KUKA KRL program: prueba_gewindebolzen_.src, prueba_gewindebolzen_.dat

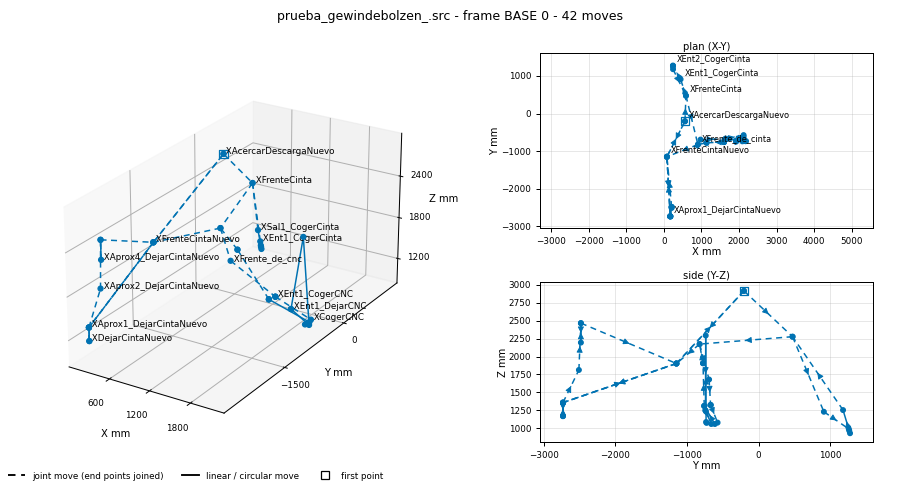
[picture p0: tool path of prueba_gewindebolzen_.src in frame BASE 0, 42 of 44 moves have a stored position in this frame; points joined in program order, loops and branches not executed]
--- prueba_gewindebolzen_.src ---
&ACCESS RVP
&REL 19
&COMMENT M36x315+allen
&PARAM TEMPLATE = C:\KRC\Roboter\Template\vorgabe
&PARAM EDITMASK = *
DEF prueba_gewindebolzen_( )
;FOLD INI;%{PE}%V3.2.0,%MKUKATPBASIS,%CINIT,%VCOMMON,%P
;FOLD BAS INI;%{E}%V3.2.0,%MKUKATPBASIS,%CINIT,%VINIT,%P
GLOBAL INTERRUPT DECL 3 WHEN $STOPMESS==TRUE DO IR_STOPM ( )
INTERRUPT ON 3
BAS (#INITMOV,0 )
;ENDFOLD (BAS INI)
;FOLD A20 INI;%{E}%V3.2.0,%MKUKATPA20,%CINIT,%VINIT,%P
IF ARC20==TRUE THEN
A20 (ARC_INI)
INTERRUPT DECL 6 WHEN $CYCFLAG[3]==FALSE DO A20(TECH_STOP2)
ENDIF
;ENDFOLD (A20 INI)
;FOLD A10 INI;%{E}%V3.2.0,%MKUKATPARC,%CINIT,%VINIT,%P
IF A10_OPTION==#ACTIVE THEN
INTERRUPT DECL 4 WHEN $CYCFLAG[2]==FALSE DO A10 (#APPL_ERROR)
INTERRUPT DECL 7 WHEN A_ARC_SWI==#ACTIVE DO A10 (#ARC_SEAM)
INTERRUPT DECL 5 WHEN A_FLY_ARC==TRUE DO A10 (#HPU_ARC)
INTERRUPT  ON 5
A10_INI ( )
ENDIF
;ENDFOLD (A10 INI)
;FOLD GRIPPER INI;%{E}%V3.2.0,%MKUKATPGRIPPER,%CINIT,%VINIT,%P
USER_GRP(0,DUMMY,DUMMY,GDEFAULT)
;ENDFOLD (GRIPPER INI)
;FOLD SPOT INI;%{E}%V3.2.0,%MKUKATPSPOT,%CINIT,%VINIT,%P
USERSPOT(#INIT)
;ENDFOLD (SPOT INI)
;FOLD TOUCHSENSE INI;%{E}%V3.2.0,%MKUKATPTS,%CINIT,%VINIT,%P
IF H70_OPTION THEN
INTERRUPT DECL 15 WHEN $MEAS_PULSE[TOUCH_I[TOUCH_ACTIVE].IN_NR] DO H70 (6,CD0 )
INTERRUPT DECL 16 WHEN $ZERO_MOVE DO H70 (7,CD0 )
INTERRUPT DECL 17 WHEN $TECHPAR_C[FG_TOUCH,8]>0.5 DO H70 (8,CD0)
H70 (1,CD0 )
ENDIF
;ENDFOLD (TOUCHSENSE INI)
;FOLD USER INI;%{E}%V3.2.0,%MKUKATPUSER,%CINIT,%VINIT,%P
;Make your modifications here
;ENDFOLD (USER INI)
;ENDFOLD (INI)

;=========================================================
;                Gewindebolzen
;       M36x315 Allen 16 + previo longitud 93
;                Codigo 257152360315
;
;=========================================================

;FOLD INICIALIZACION

INTERRUPT DECL 20 WHEN $IN[20]==FALSE DO PARO()
INTERRUPT OFF 20
;FOLD WAIT FOR IN 20 'InAire'  State= TRUE ;%{PE}%R 4.1.7,%MKUKATPBASIS,%CWAIT_FOR,%VWAIT_FOR,%P 1:0, 2:20, 3:'InAire', 5:TRUE, 6:
WAIT FOR $IN[20]==TRUE
;ENDFOLD


;FOLD PTP HOME CONT Vel= 5 % PDAT1;%{PE}%R 4.1.7,%MKUKATPBASIS,%CMOVE,%VPTP,%P 1:PTP, 2:HOME, 3:C_PTP, 5:5, 7:PDAT1
$BWDSTART = FALSE
PDAT_ACT=PPDAT1
BAS(#PTP_DAT)
FDAT_ACT=FHOME
BAS(#FRAMES)
BAS(#VEL_PTP,5)
$H_POS=XHOME
PTP XHOME C_PTP
;ENDFOLD
;FOLD WAIT Time=0 sec;%{PE}%R 5.5.32,%MKUKATPBASIS,%CWAIT,%VWAIT,%P 2:0
WAIT SEC 0
;ENDFOLD
DELMENS()


INTERRUPT ON 20

;$OV_PRO=nVeloFuera

bMarchaCintaSuperior=FALSE
bRobotEnCintaSup=FALSE
;FOLD OUT 1 'OutMarchaCintaSup'  State= FALSE CONT;%{PE}%R 4.1.7,%MKUKATPBASIS,%COUT,%VOUTX,%P 2:1, 3:'OutMarchaCintaSup', 5:FALSE, 6:CONTINUE
CONTINUE
$OUT[1]=FALSE
;ENDFOLD
;FOLD OUT 2 'OutMarchaCNC'  State= FALSE CONT;%{PE}%R 4.1.7,%MKUKATPBASIS,%COUT,%VOUTX,%P 2:2, 3:'OutMarchaCNC', 5:FALSE, 6:CONTINUE
CONTINUE
$OUT[2]=FALSE
;ENDFOLD
;FOLD OUT 3 'OutRobotDentroCNC'  State= FALSE CONT;%{PE}%R 4.1.7,%MKUKATPBASIS,%COUT,%VOUTX,%P 2:3, 3:'OutRobotDentroCNC', 5:FALSE, 6:CONTINUE
CONTINUE
$OUT[3]=FALSE
;ENDFOLD
;FOLD OUT 7 'OutRobotFuerCNC'  State= TRUE CONT;%{PE}%R 4.1.7,%MKUKATPBASIS,%COUT,%VOUTX,%P 2:7, 3:'OutRobotFuerCNC', 5:TRUE, 6:CONTINUE
CONTINUE
$OUT[7]=TRUE
;ENDFOLD
;FOLD OUT 8 'OutAbrirPlatoCNC'  State= FALSE CONT;%{PE}%R 4.1.7,%MKUKATPBASIS,%COUT,%VOUTX,%P 2:8, 3:'OutAbrirPlatoCNC', 5:FALSE, 6:CONTINUE
CONTINUE
$OUT[8]=FALSE
;ENDFOLD
;FOLD OUT 9 'OutCerrarPlatoCNC'  State= FALSE CONT;%{PE}%R 4.1.7,%MKUKATPBASIS,%COUT,%VOUTX,%P 2:9, 3:'OutCerrarPlatoCNC', 5:FALSE, 6:CONTINUE
CONTINUE
$OUT[9]=FALSE
;ENDFOLD
;FOLD OUT 10 'OutAvanContrpuntoCNC'  State= FALSE CONT;%{PE}%R 4.1.7,%MKUKATPBASIS,%COUT,%VOUTX,%P 2:10, 3:'OutAvanContrpuntoCNC', 5:FALSE, 6:CONTINUE
CONTINUE
$OUT[10]=FALSE
;ENDFOLD
;FOLD OUT 11 'OutRetroContrpuntoCNC'  State= FALSE CONT;%{PE}%R 4.1.7,%MKUKATPBASIS,%COUT,%VOUTX,%P 2:11, 3:'OutRetroContrpuntoCNC', 5:FALSE, 6:CONTINUE
CONTINUE
$OUT[11]=FALSE
;ENDFOLD
;FOLD OUT 12 'OutAbrirLunetaCNC'  State= FALSE CONT;%{PE}%R 4.1.7,%MKUKATPBASIS,%COUT,%VOUTX,%P 2:12, 3:'OutAbrirLunetaCNC', 5:FALSE, 6:CONTINUE
CONTINUE
$OUT[12]=FALSE
;ENDFOLD
;FOLD OUT 17 'OutCerrarLunetaCNC'  State= FALSE CONT;%{PE}%R 4.1.7,%MKUKATPBASIS,%COUT,%VOUTX,%P 2:17, 3:'OutCerrarLunetaCNC', 5:FALSE, 6:CONTINUE
CONTINUE
$OUT[17]=FALSE
;ENDFOLD


bParadaManiobra=FALSE
;FOLD WAIT FOR ( IN 4 'InPulsadorMarcha' );%{PE}%R 5.5.33,%MKUKATPBASIS,%CEXT_WAIT_FOR,%VEXT_WAIT_FOR,%P 2:, 4:, 5:$IN, 6:4, 7:InPulsadorMarcha, 9:
WAIT FOR  ( $IN[4] )
;ENDFOLD
bMarchaCintaSuperior=TRUE
;FOLD WAIT Time=0.5 sec;%{PE}%R 5.5.33,%MKUKATPBASIS,%CWAIT,%VWAIT,%P 2:0.5
WAIT SEC 0.5
;ENDFOLD
bMarchaCintaSuperior=FALSE
;FOLD WAIT FOR NOT ( IN 4 'InPulsadorMarcha' );%{PE}%R 5.5.33,%MKUKATPBASIS,%CEXT_WAIT_FOR,%VEXT_WAIT_FOR,%P 2:NOT, 4:, 5:$IN, 6:4, 7:InPulsadorMarcha, 9:
WAIT FOR  NOT ( $IN[4] )
;ENDFOLD
outPilotoMarcha=TRUE

;------Soltar Piezas sobre Cinta de Descarga-------
IF ((InPinza1Abierta==FALSE) OR (InPinza2Abierta==FALSE)) THEN


;FOLD PTP AcercarDescargaNuevo CONT Vel= 30 % PDAT28 Tool[0] Base[0];%{PE}%R 4.1.16,%MKUKATPBASIS,%CMOVE,%VPTP,%P 1:PTP, 2:AcercarDescargaNuevo, 3:C_PTP, 5:30, 7:PDAT28
$BWDSTART = FALSE
PDAT_ACT=PPDAT28
BAS(#PTP_DAT)
FDAT_ACT=FAcercarDescargaNuevo
BAS(#FRAMES)
BAS(#VEL_PTP,30)
PTP XAcercarDescargaNuevo C_PTP
;ENDFOLD

;FOLD PTP FrenteCintaNuevo CONT Vel= 30 % PDAT26 Tool[0] Base[0];%{PE}%R 4.1.16,%MKUKATPBASIS,%CMOVE,%VPTP,%P 1:PTP, 2:FrenteCintaNuevo, 3:C_PTP, 5:30, 7:PDAT26
$BWDSTART = FALSE
PDAT_ACT=PPDAT26
BAS(#PTP_DAT)
FDAT_ACT=FFrenteCintaNuevo
BAS(#FRAMES)
BAS(#VEL_PTP,30)
PTP XFrenteCintaNuevo C_PTP
;ENDFOLD

;FOLD PTP Aprox1_DejarCintaNuevo CONT Vel= 30 % PDAT27 Tool[2]:Tool2      Base[0];%{PE}%R 4.1.16,%MKUKATPBASIS,%CMOVE,%VPTP,%P 1:PTP, 2:Aprox1_DejarCintaNuevo, 3:C_PTP, 5:30, 7:PDAT27
$BWDSTART = FALSE
PDAT_ACT=PPDAT27
BAS(#PTP_DAT)
FDAT_ACT=FAprox1_DejarCintaNuevo
BAS(#FRAMES)
BAS(#VEL_PTP,30)
PTP XAprox1_DejarCintaNuevo C_PTP
;ENDFOLD

;FOLD LIN DejarCintaNuevo CONT Vel= 0.3 m/s CPDAT1 Tool[2]:Tool2      Base[0];%{PE}%R 4.1.16,%MKUKATPBASIS,%CMOVE,%VLIN,%P 1:LIN, 2:DejarCintaNuevo, 3:C_DIS, 5:0.3, 7:CPDAT1
$BWDSTART = FALSE
LDAT_ACT=LCPDAT1
BAS(#CP_DAT)
FDAT_ACT=FDejarCintaNuevo
BAS(#FRAMES)
BAS(#VEL_CP,0.3)
LIN XDejarCintaNuevo C_DIS
;ENDFOLD

;FOLD SET Pinza2  State= OPN  Abrir;%{PE}%R 4.1.4,%MKUKATPGRP,%CGRP,%VGRP,%P 2:2, 4:1, 5:#NO, 6:Abrir, 8:0, 10:1
H50(GRP,2,1,GAbrir)
;ENDFOLD

;FOLD PTP Aprox1_DejarCintaNuevo CONT Vel= 30 % PDAT27 Tool[2]:Tool2      Base[0];%{PE}%R 4.1.16,%MKUKATPBASIS,%CMOVE,%VPTP,%P 1:PTP, 2:Aprox1_DejarCintaNuevo, 3:C_PTP, 5:30, 7:PDAT27
$BWDSTART = FALSE
PDAT_ACT=PPDAT27
BAS(#PTP_DAT)
FDAT_ACT=FAprox1_DejarCintaNuevo
BAS(#FRAMES)
BAS(#VEL_PTP,30)
PTP XAprox1_DejarCintaNuevo C_PTP
;ENDFOLD

;FOLD PTP Aprox2_DejarCintaNuevo CONT Vel= 30 % PDAT29 Tool[2]:Tool2      Base[0];%{PE}%R 4.1.16,%MKUKATPBASIS,%CMOVE,%VPTP,%P 1:PTP, 2:Aprox2_DejarCintaNuevo, 3:C_PTP, 5:30, 7:PDAT29
$BWDSTART = FALSE
PDAT_ACT=PPDAT29
BAS(#PTP_DAT)
FDAT_ACT=FAprox2_DejarCintaNuevo
BAS(#FRAMES)
BAS(#VEL_PTP,30)
PTP XAprox2_DejarCintaNuevo C_PTP
;ENDFOLD

;FOLD PTP Aprox3_DejarCintaNuevo CONT Vel= 30 % PDAT30 Tool[2]:Tool2      Base[0];%{PE}%R 4.1.16,%MKUKATPBASIS,%CMOVE,%VPTP,%P 1:PTP, 2:Aprox3_DejarCintaNuevo, 3:C_PTP, 5:30, 7:PDAT30
$BWDSTART = FALSE
PDAT_ACT=PPDAT30
BAS(#PTP_DAT)
FDAT_ACT=FAprox3_DejarCintaNuevo
BAS(#FRAMES)
BAS(#VEL_PTP,30)
PTP XAprox3_DejarCintaNuevo C_PTP
;ENDFOLD

;FOLD LIN Aprox4_DejarCintaNuevo CONT Vel= 0.3 m/s CPDAT13 Tool[2]:Tool2      Base[0];%{PE}%R 4.1.16,%MKUKATPBASIS,%CMOVE,%VLIN,%P 1:LIN, 2:Aprox4_DejarCintaNuevo, 3:C_DIS, 5:0.3, 7:CPDAT13
$BWDSTART = FALSE
LDAT_ACT=LCPDAT13
BAS(#CP_DAT)
FDAT_ACT=FAprox4_DejarCintaNuevo
BAS(#FRAMES)
BAS(#VEL_CP,0.3)
LIN XAprox4_DejarCintaNuevo C_DIS
;ENDFOLD

;FOLD SET Pinza1  State= OPN  Abrir;%{PE}%R 4.1.4,%MKUKATPGRP,%CGRP,%VGRP,%P 2:1, 4:1, 5:#NO, 6:Abrir, 8:0, 10:1
H50(GRP,1,1,GAbrir)
;ENDFOLD

;FOLD PTP Aprox3_DejarCintaNuevo CONT Vel= 30 % PDAT30 Tool[2]:Tool2      Base[0];%{PE}%R 4.1.16,%MKUKATPBASIS,%CMOVE,%VPTP,%P 1:PTP, 2:Aprox3_DejarCintaNuevo, 3:C_PTP, 5:30, 7:PDAT30
$BWDSTART = FALSE
PDAT_ACT=PPDAT30
BAS(#PTP_DAT)
FDAT_ACT=FAprox3_DejarCintaNuevo
BAS(#FRAMES)
BAS(#VEL_PTP,30)
PTP XAprox3_DejarCintaNuevo C_PTP
;ENDFOLD

;FOLD PTP FrenteCintaNuevo CONT Vel= 30 % PDAT26 Tool[0] Base[0];%{PE}%R 4.1.16,%MKUKATPBASIS,%CMOVE,%VPTP,%P 1:PTP, 2:FrenteCintaNuevo, 3:C_PTP, 5:30, 7:PDAT26
$BWDSTART = FALSE
PDAT_ACT=PPDAT26
BAS(#PTP_DAT)
FDAT_ACT=FFrenteCintaNuevo
BAS(#FRAMES)
BAS(#VEL_PTP,30)
PTP XFrenteCintaNuevo C_PTP
;ENDFOLD

;FOLD PTP AcercarDescargaNuevo CONT Vel= 30 % PDAT28 Tool[0] Base[0];%{PE}%R 4.1.16,%MKUKATPBASIS,%CMOVE,%VPTP,%P 1:PTP, 2:AcercarDescargaNuevo, 3:C_PTP, 5:30, 7:PDAT28
$BWDSTART = FALSE
PDAT_ACT=PPDAT28
BAS(#PTP_DAT)
FDAT_ACT=FAcercarDescargaNuevo
BAS(#FRAMES)
BAS(#VEL_PTP,30)
PTP XAcercarDescargaNuevo C_PTP
;ENDFOLD

ELSE

ENDIF

LOOP


;FOLD CHECK Pinza1  State= OPN  at START  Delay= 0 ms;%{PE}%R 4.1.4,%MKUKATPGRP,%CCHK_GRP,%VCHK_GRP,%P 2:1, 4:1, 6:0, 8:0
TRIGGER WHEN DISTANCE=0 DELAY=0 DO H50(CHK_APO_UP,1,1,GCONT)  PRIO=-1
;ENDFOLD
;FOLD CHECK Pinza2  State= OPN  at START  Delay= 0 ms;%{PE}%R 4.1.4,%MKUKATPGRP,%CCHK_GRP,%VCHK_GRP,%P 2:2, 4:1, 6:0, 8:0
TRIGGER WHEN DISTANCE=0 DELAY=0 DO H50(CHK_APO_UP,2,1,GCONT)  PRIO=-1
;ENDFOLD

;FOLD WAIT FOR IN 21 'InPinza1Abierta'  State= TRUE ;%{PE}%R 4.1.7,%MKUKATPBASIS,%CWAIT_FOR,%VWAIT_FOR,%P 1:0, 2:21, 3:'InPinza1Abierta', 5:TRUE, 6:
WAIT FOR $IN[21]==TRUE
;ENDFOLD
;FOLD WAIT FOR IN 23 'InPinza2Abierta'  State= TRUE ;%{PE}%R 4.1.7,%MKUKATPBASIS,%CWAIT_FOR,%VWAIT_FOR,%P 1:0, 2:23, 3:'InPinza2Abierta', 5:TRUE, 6:
WAIT FOR $IN[23]==TRUE
;ENDFOLD
;ENDFOLD


;FOLD COGER PIEZA DE CINTA

;FOLD PTP FrenteCinta CONT Vel= 30 % PDAT1 Tool[0] Base[0];%{PE}%R 4.1.7,%MKUKATPBASIS,%CMOVE,%VPTP,%P 1:PTP, 2:FrenteCinta, 3:C_PTP, 5:30, 7:PDAT1
$BWDSTART = FALSE
PDAT_ACT=PPDAT1
BAS(#PTP_DAT)
FDAT_ACT=FFrenteCinta
BAS(#FRAMES)
BAS(#VEL_PTP,30)
PTP XFrenteCinta C_PTP
;ENDFOLD

;FOLD PTP Ent1_CogerCinta CONT Vel= 30 % PDAT1 Tool[1]:Tool1      Base[0];%{PE}%R 4.1.7,%MKUKATPBASIS,%CMOVE,%VPTP,%P 1:PTP, 2:Ent1_CogerCinta, 3:C_PTP, 5:30, 7:PDAT1
$BWDSTART = FALSE
PDAT_ACT=PPDAT1
BAS(#PTP_DAT)
FDAT_ACT=FEnt1_CogerCinta
BAS(#FRAMES)
BAS(#VEL_PTP,30)
PTP XEnt1_CogerCinta C_PTP
;ENDFOLD

WAIT FOR ($IN[11] AND $IN[12])


;FOLD PTP Ent2_CogerCinta CONT Vel= 30 % PDAT1 Tool[1]:Tool1      Base[0];%{PE}%R 4.1.7,%MKUKATPBASIS,%CMOVE,%VPTP,%P 1:PTP, 2:Ent2_CogerCinta, 3:C_PTP, 5:30, 7:PDAT1
$BWDSTART = FALSE
PDAT_ACT=PPDAT1
BAS(#PTP_DAT)
FDAT_ACT=FEnt2_CogerCinta
BAS(#FRAMES)
BAS(#VEL_PTP,30)
PTP XEnt2_CogerCinta C_PTP
;ENDFOLD
bRobotEnCintaSup=TRUE

;FOLD LIN Ent3CogerCinta CONT Vel= 0.3 m/s CPDAT1 Tool[1]:Tool1      Base[0];%{PE}%R 4.1.7,%MKUKATPBASIS,%CMOVE,%VLIN,%P 1:LIN, 2:Ent3CogerCinta, 3:C_DIS, 5:0.3, 7:CPDAT1
$BWDSTART = FALSE
LDAT_ACT=LCPDAT1
BAS(#CP_DAT)
FDAT_ACT=FEnt3CogerCinta
BAS(#FRAMES)
BAS(#VEL_CP,0.3)
LIN XEnt3CogerCinta C_DIS
;ENDFOLD
;FOLD LIN CogerCinta CONT Vel= 2 m/s CPDAT1 Tool[1]:Tool1      Base[0];%{PE}%R 4.1.7,%MKUKATPBASIS,%CMOVE,%VLIN,%P 1:LIN, 2:CogerCinta, 3:C_DIS, 5:2, 7:CPDAT1
$BWDSTART = FALSE
LDAT_ACT=LCPDAT1
BAS(#CP_DAT)
FDAT_ACT=FCogerCinta
BAS(#FRAMES)
BAS(#VEL_CP,2)
LIN XCogerCinta C_DIS
;ENDFOLD

;FOLD SET Pinza1  State= CLO  Cerrar;%{PE}%R 4.1.4,%MKUKATPGRP,%CGRP,%VGRP,%P 2:1, 4:2, 5:#NO, 6:Cerrar, 8:0, 10:1
H50(GRP,1,2,GCerrar)
;ENDFOLD

;FOLD LIN Sal1_CogerCinta  Vel= 0.5 m/s CPDAT1 Tool[1]:Tool1      Base[0];%{PE}%R 4.1.7,%MKUKATPBASIS,%CMOVE,%VLIN,%P 1:LIN, 2:Sal1_CogerCinta, 3:, 5:0.5, 7:CPDAT1
$BWDSTART = FALSE
LDAT_ACT=LCPDAT1
BAS(#CP_DAT)
FDAT_ACT=FSal1_CogerCinta
BAS(#FRAMES)
BAS(#VEL_CP,0.5)
LIN XSal1_CogerCinta
;ENDFOLD
$advance=1
bRobotEnCintaSup=FALSE
;FOLD WAIT Time= 2 sec;%{PE}%R 4.1.16,%MKUKATPBASIS,%CWAIT,%VWAIT,%P 2:2
WAIT SEC 2
;ENDFOLD
bMarchaCintaSuperior=TRUE
;FOLD PTP FrenteCinta CONT Vel= 30 % PDAT1 Tool[0] Base[0];%{PE}%R 4.1.7,%MKUKATPBASIS,%CMOVE,%VPTP,%P 1:PTP, 2:FrenteCinta, 3:C_PTP, 5:30, 7:PDAT1
$BWDSTART = FALSE
PDAT_ACT=PPDAT1
BAS(#PTP_DAT)
FDAT_ACT=FFrenteCinta
BAS(#FRAMES)
BAS(#VEL_PTP,30)
PTP XFrenteCinta C_PTP
;ENDFOLD

;FOLD WAIT Time= 0.5 sec;%{PE}%R 4.1.7,%MKUKATPBASIS,%CWAIT,%VWAIT,%P 2:0.5
WAIT SEC 0.5
;ENDFOLD
bMarchaCintaSuperior=FALSE
$advance=3

;ENDFOLD
;FOLD CARGA/DESCARGA DE CNC

;FOLD PTP Frente_de_cinta CONT Vel= 50 % PDAT21 Tool[0] Base[0];%{PE}%R 4.1.7,%MKUKATPBASIS,%CMOVE,%VPTP,%P 1:PTP, 2:Frente_de_cinta, 3:C_PTP, 5:50, 7:PDAT21
$BWDSTART = FALSE
PDAT_ACT=PPDAT21
BAS(#PTP_DAT)
FDAT_ACT=FFrente_de_cinta
BAS(#FRAMES)
BAS(#VEL_PTP,50)
PTP XFrente_de_cinta C_PTP
;ENDFOLD

;FOLD PTP Frente_de_cnc CONT Vel= 50 % PDAT1 Tool[0] Base[0];%{PE}%R 4.1.7,%MKUKATPBASIS,%CMOVE,%VPTP,%P 1:PTP, 2:Frente_de_cnc, 3:C_PTP, 5:50, 7:PDAT1
$BWDSTART = FALSE
PDAT_ACT=PPDAT1
BAS(#PTP_DAT)
FDAT_ACT=FFrente_de_cnc
BAS(#FRAMES)
BAS(#VEL_PTP,50)
PTP XFrente_de_cnc C_PTP
;ENDFOLD

;FOLD WAIT FOR IN 18 'InPermRobCargaCNC'  State= TRUE ;%{PE}%R 4.1.7,%MKUKATPBASIS,%CWAIT_FOR,%VWAIT_FOR,%P 1:0, 2:18, 3:'InPermRobCargaCNC', 5:TRUE, 6:
WAIT FOR $IN[18]==TRUE
;ENDFOLD
;FOLD WAIT FOR IN 19 'InNoAlarmasCNC'  State= TRUE ;%{PE}%R 4.1.7,%MKUKATPBASIS,%CWAIT_FOR,%VWAIT_FOR,%P 1:0, 2:19, 3:'InNoAlarmasCNC', 5:TRUE, 6:
WAIT FOR $IN[19]==TRUE
;ENDFOLD
;FOLD WAIT FOR IN 25 'InConRobotCNC'  State= TRUE ;%{PE}%R 4.1.7,%MKUKATPBASIS,%CWAIT_FOR,%VWAIT_FOR,%P 1:0, 2:25, 3:'InConRobotCNC', 5:TRUE, 6:
WAIT FOR $IN[25]==TRUE
;ENDFOLD
;FOLD WAIT FOR IN 26 'InPuertaAbiertaCNC'  State= TRUE ;%{PE}%R 4.1.7,%MKUKATPBASIS,%CWAIT_FOR,%VWAIT_FOR,%P 1:0, 2:26, 3:'InPuertaAbiertaCNC', 5:TRUE, 6:
WAIT FOR $IN[26]==TRUE
;ENDFOLD

WAIT FOR $IN[18] AND $IN[19] AND $IN[25] AND $IN[26]

;FOLD OUT 3 'OutRobotDentroCNC'  State= TRUE ;%{PE}%R 4.1.7,%MKUKATPBASIS,%COUT,%VOUTX,%P 2:3, 3:'OutRobotDentroCNC', 5:TRUE, 6:
$OUT[3]=TRUE
;ENDFOLD
;FOLD OUT 7 'OutRobotFuerCNC'  State= FALSE ;%{PE}%R 4.1.7,%MKUKATPBASIS,%COUT,%VOUTX,%P 2:7, 3:'OutRobotFuerCNC', 5:FALSE, 6:
$OUT[7]=FALSE
;ENDFOLD


;------------Coger Pieza de CNC-------------

;FOLD PTP Ent1_CogerCNC CONT Vel= 100 % PDAT1 Tool[2]:Tool2      Base[0];%{PE}%R 4.1.7,%MKUKATPBASIS,%CMOVE,%VPTP,%P 1:PTP, 2:Ent1_CogerCNC, 3:C_PTP, 5:100, 7:PDAT1
$BWDSTART = FALSE
PDAT_ACT=PPDAT1
BAS(#PTP_DAT)
FDAT_ACT=FEnt1_CogerCNC
BAS(#FRAMES)
BAS(#VEL_PTP,100)
PTP XEnt1_CogerCNC C_PTP
;ENDFOLD

;FOLD WAIT FOR IN 18 'InPermRobCargaCNC'  State= TRUE ;%{PE}%R 4.1.7,%MKUKATPBASIS,%CWAIT_FOR,%VWAIT_FOR,%P 1:0, 2:18, 3:'InPermRobCargaCNC', 5:TRUE, 6:
WAIT FOR $IN[18]==TRUE
;ENDFOLD
;FOLD WAIT FOR IN 19 'InNoAlarmasCNC'  State= TRUE ;%{PE}%R 4.1.7,%MKUKATPBASIS,%CWAIT_FOR,%VWAIT_FOR,%P 1:0, 2:19, 3:'InNoAlarmasCNC', 5:TRUE, 6:
WAIT FOR $IN[19]==TRUE
;ENDFOLD
;FOLD WAIT FOR IN 25 'InConRobotCNC'  State= TRUE ;%{PE}%R 4.1.7,%MKUKATPBASIS,%CWAIT_FOR,%VWAIT_FOR,%P 1:0, 2:25, 3:'InConRobotCNC', 5:TRUE, 6:
WAIT FOR $IN[25]==TRUE
;ENDFOLD
;FOLD WAIT FOR IN 26 'InPuertaAbiertaCNC'  State= TRUE ;%{PE}%R 4.1.7,%MKUKATPBASIS,%CWAIT_FOR,%VWAIT_FOR,%P 1:0, 2:26, 3:'InPuertaAbiertaCNC', 5:TRUE, 6:
WAIT FOR $IN[26]==TRUE
;ENDFOLD

WAIT FOR $IN[18] AND $IN[19] AND $IN[25] AND $IN[26]


;FOLD TORQMON.SetLimits Axis 1: 50 %, Axis 2: 50 %, Axis 3: 50 %, Axis 4: 50 %, Axis 5: 50 %, Axis 6: 50 %;%{PE}%MKUKATPUSER
$TORQMON[1]=50
$TORQMON[2]=50
$TORQMON[3]=50
$TORQMON[4]=50
$TORQMON[5]=50
$TORQMON[6]=50
;ENDFOLD

;FOLD PTP Ent2_CogerCNC CONT Vel= 100 % PDAT1 Tool[2]:Tool2      Base[0];%{PE}%R 4.1.7,%MKUKATPBASIS,%CMOVE,%VPTP,%P 1:PTP, 2:Ent2_CogerCNC, 3:C_PTP, 5:100, 7:PDAT1
$BWDSTART = FALSE
PDAT_ACT=PPDAT1
BAS(#PTP_DAT)
FDAT_ACT=FEnt2_CogerCNC
BAS(#FRAMES)
BAS(#VEL_PTP,100)
PTP XEnt2_CogerCNC C_PTP
;ENDFOLD
;FOLD LIN Ent3_CogerCNC CONT Vel= 2 m/s CPDAT1 Tool[2]:Tool2      Base[0];%{PE}%R 4.1.7,%MKUKATPBASIS,%CMOVE,%VLIN,%P 1:LIN, 2:Ent3_CogerCNC, 3:C_DIS, 5:2, 7:CPDAT1
$BWDSTART = FALSE
LDAT_ACT=LCPDAT1
BAS(#CP_DAT)
FDAT_ACT=FEnt3_CogerCNC
BAS(#FRAMES)
BAS(#VEL_CP,2)
LIN XEnt3_CogerCNC C_DIS
;ENDFOLD
;FOLD PTP CogerCNC CONT Vel= 100 % PDAT22 Tool[2]:Tool2      Base[0];%{PE}%R 4.1.7,%MKUKATPBASIS,%CMOVE,%VPTP,%P 1:PTP, 2:CogerCNC, 3:C_PTP, 5:100, 7:PDAT22
$BWDSTART = FALSE
PDAT_ACT=PPDAT22
BAS(#PTP_DAT)
FDAT_ACT=FCogerCNC
BAS(#FRAMES)
BAS(#VEL_PTP,100)
PTP XCogerCNC C_PTP
;ENDFOLD
;FOLD WAIT Time=0 sec;%{PE}%R 5.5.33,%MKUKATPBASIS,%CWAIT,%VWAIT,%P 2:0
WAIT SEC 0
;ENDFOLD

;FOLD SET Pinza2  State= CLO  Cerrar;%{PE}%R 4.1.4,%MKUKATPGRP,%CGRP,%VGRP,%P 2:2, 4:2, 5:#NO, 6:Cerrar, 8:0, 10:1
H50(GRP,2,2,GCerrar)
;ENDFOLD

;--Retroceso contrapunto--
;FOLD OUT 10 'OutAvanContrpuntoCNC'  State= FALSE ;%{PE}%R 4.1.7,%MKUKATPBASIS,%COUT,%VOUTX,%P 2:10, 3:'OutAvanContrpuntoCNC', 5:FALSE, 6:
$OUT[10]=FALSE
;ENDFOLD
;FOLD OUT 11 'OutRetroContrpuntoCNC'  State= TRUE ;%{PE}%R 4.1.7,%MKUKATPBASIS,%COUT,%VOUTX,%P 2:11, 3:'OutRetroContrpuntoCNC', 5:TRUE, 6:
$OUT[11]=TRUE
;ENDFOLD
;--Abrir Luneta---
;FOLD OUT 12 'OutAbrirLunetaCNC'  State= TRUE CONT;%{PE}%R 4.1.7,%MKUKATPBASIS,%COUT,%VOUTX,%P 2:12, 3:'OutAbrirLunetaCNC', 5:TRUE, 6:CONTINUE
CONTINUE
$OUT[12]=TRUE
;ENDFOLD
;FOLD OUT 17 'OutCerrarLunetaCNC'  State= FALSE CONT;%{PE}%R 4.1.7,%MKUKATPBASIS,%COUT,%VOUTX,%P 2:17, 3:'OutCerrarLunetaCNC', 5:FALSE, 6:CONTINUE
CONTINUE
$OUT[17]=FALSE
;ENDFOLD
;--Abrir Plato
;FOLD OUT 8 'OutAbrirPlatoCNC'  State= TRUE CONT;%{PE}%R 4.1.7,%MKUKATPBASIS,%COUT,%VOUTX,%P 2:8, 3:'OutAbrirPlatoCNC', 5:TRUE, 6:CONTINUE
CONTINUE
$OUT[8]=TRUE
;ENDFOLD
;FOLD OUT 9 'OutCerrarPlatoCNC'  State= FALSE CONT;%{PE}%R 4.1.7,%MKUKATPBASIS,%COUT,%VOUTX,%P 2:9, 3:'OutCerrarPlatoCNC', 5:FALSE, 6:CONTINUE
CONTINUE
$OUT[9]=FALSE
;ENDFOLD

;FOLD WAIT FOR IN 13 'InContrpuntoAtrasCNC'  State= TRUE ;%{PE}%R 4.1.7,%MKUKATPBASIS,%CWAIT_FOR,%VWAIT_FOR,%P 1:0, 2:13, 3:'InContrpuntoAtrasCNC', 5:TRUE, 6:
WAIT FOR $IN[13]==TRUE
;ENDFOLD
;FOLD OUT 11 'OutRetroContrpuntoCNC'  State= FALSE ;%{PE}%R 4.1.7,%MKUKATPBASIS,%COUT,%VOUTX,%P 2:11, 3:'OutRetroContrpuntoCNC', 5:FALSE, 6:
$OUT[11]=FALSE
;ENDFOLD
;-----------------------
;FOLD WAIT FOR IN 16 'InLunetaAbiertaCNC'  State= TRUE ;%{PE}%R 4.1.7,%MKUKATPBASIS,%CWAIT_FOR,%VWAIT_FOR,%P 1:0, 2:16, 3:'InLunetaAbiertaCNC', 5:TRUE, 6:
WAIT FOR $IN[16]==TRUE
;ENDFOLD
;FOLD OUT 12 'OutAbrirLunetaCNC'  State= FALSE ;%{PE}%R 4.1.7,%MKUKATPBASIS,%COUT,%VOUTX,%P 2:12, 3:'OutAbrirLunetaCNC', 5:FALSE, 6:
$OUT[12]=FALSE
;ENDFOLD
;--------------------
;FOLD WAIT FOR IN 14 'InPlatoAbiertoCNC'  State= TRUE ;%{PE}%R 4.1.7,%MKUKATPBASIS,%CWAIT_FOR,%VWAIT_FOR,%P 1:0, 2:14, 3:'InPlatoAbiertoCNC', 5:TRUE, 6:
WAIT FOR $IN[14]==TRUE
;ENDFOLD
;FOLD OUT 8 'OutAbrirPlatoCNC'  State= FALSE ;%{PE}%R 4.1.7,%MKUKATPBASIS,%COUT,%VOUTX,%P 2:8, 3:'OutAbrirPlatoCNC', 5:FALSE, 6:
$OUT[8]=FALSE
;ENDFOLD
;FOLD WAIT Time= 0 sec;%{PE}%R 4.1.7,%MKUKATPBASIS,%CWAIT,%VWAIT,%P 2:0
WAIT SEC 0
;ENDFOLD
;-------------------

;FOLD LIN Sal1_CogerCNC  Vel= 2 m/s CPDAT1 Tool[2]:Tool2      Base[0];%{PE}%R 4.1.7,%MKUKATPBASIS,%CMOVE,%VLIN,%P 1:LIN, 2:Sal1_CogerCNC, 3:, 5:2, 7:CPDAT1
$BWDSTART = FALSE
LDAT_ACT=LCPDAT1
BAS(#CP_DAT)
FDAT_ACT=FSal1_CogerCNC
BAS(#FRAMES)
BAS(#VEL_CP,2)
LIN XSal1_CogerCNC
;ENDFOLD
;FOLD LIN Sal2_CogerCNC CONT Vel= 2 m/s CPDAT1 Tool[2]:Tool2      Base[0];%{PE}%R 4.1.7,%MKUKATPBASIS,%CMOVE,%VLIN,%P 1:LIN, 2:Sal2_CogerCNC, 3:C_DIS, 5:2, 7:CPDAT1
$BWDSTART = FALSE
LDAT_ACT=LCPDAT1
BAS(#CP_DAT)
FDAT_ACT=FSal2_CogerCNC
BAS(#FRAMES)
BAS(#VEL_CP,2)
LIN XSal2_CogerCNC C_DIS
;ENDFOLD
;FOLD LIN Sal3_CojerCNC CONT Vel= 2 m/s CPDAT1 Tool[2]:Tool2      Base[0];%{PE}%R 4.1.7,%MKUKATPBASIS,%CMOVE,%VLIN,%P 1:LIN, 2:Sal3_CojerCNC, 3:C_DIS, 5:2, 7:CPDAT1
$BWDSTART = FALSE
LDAT_ACT=LCPDAT1
BAS(#CP_DAT)
FDAT_ACT=FSal3_CojerCNC
BAS(#FRAMES)
BAS(#VEL_CP,2)
LIN XSal3_CojerCNC C_DIS
;ENDFOLD


;------------Dejar Pieza en CNC-------------

;FOLD LIN Ent1_DejarCNC CONT Vel= 2 m/s CPDAT1 Tool[1]:Tool1      Base[0];%{PE}%R 4.1.7,%MKUKATPBASIS,%CMOVE,%VLIN,%P 1:LIN, 2:Ent1_DejarCNC, 3:C_DIS, 5:2, 7:CPDAT1
$BWDSTART = FALSE
LDAT_ACT=LCPDAT1
BAS(#CP_DAT)
FDAT_ACT=FEnt1_DejarCNC
BAS(#FRAMES)
BAS(#VEL_CP,2)
LIN XEnt1_DejarCNC C_DIS
;ENDFOLD
;FOLD LIN Ent2_DejarCNC CONT Vel= 2 m/s CPDAT1 Tool[1]:Tool1      Base[0];%{PE}%R 4.1.7,%MKUKATPBASIS,%CMOVE,%VLIN,%P 1:LIN, 2:Ent2_DejarCNC, 3:C_DIS, 5:2, 7:CPDAT1
$BWDSTART = FALSE
LDAT_ACT=LCPDAT1
BAS(#CP_DAT)
FDAT_ACT=FEnt2_DejarCNC
BAS(#FRAMES)
BAS(#VEL_CP,2)
LIN XEnt2_DejarCNC C_DIS
;ENDFOLD
;FOLD LIN Ent3_DejarCNC  Vel= 2 m/s CPDAT1 Tool[1]:Tool1      Base[0];%{PE}%R 4.1.7,%MKUKATPBASIS,%CMOVE,%VLIN,%P 1:LIN, 2:Ent3_DejarCNC, 3:, 5:2, 7:CPDAT1
$BWDSTART = FALSE
LDAT_ACT=LCPDAT1
BAS(#CP_DAT)
FDAT_ACT=FEnt3_DejarCNC
BAS(#FRAMES)
BAS(#VEL_CP,2)
LIN XEnt3_DejarCNC
;ENDFOLD
;FOLD LIN DejarCNC  Vel= 2 m/s CPDAT1 Tool[1]:Tool1      Base[0];%{PE}%R 4.1.7,%MKUKATPBASIS,%CMOVE,%VLIN,%P 1:LIN, 2:DejarCNC, 3:, 5:2, 7:CPDAT1
$BWDSTART = FALSE
LDAT_ACT=LCPDAT1
BAS(#CP_DAT)
FDAT_ACT=FDejarCNC
BAS(#FRAMES)
BAS(#VEL_CP,2)
LIN XDejarCNC
;ENDFOLD
;FOLD WAIT Time=0 sec;%{PE}%R 5.5.33,%MKUKATPBASIS,%CWAIT,%VWAIT,%P 2:0
WAIT SEC 0
;ENDFOLD

;--Avanzar Contrapunto--
;FOLD OUT 10 'OutAvanContrpuntoCNC'  State= FALSE ;%{PE}%R 4.1.16,%MKUKATPBASIS,%COUT,%VOUTX,%P 2:10, 3:'OutAvanContrpuntoCNC', 5:FALSE, 6:
$OUT[10]=FALSE
;ENDFOLD
;FOLD OUT 11 'OutRetroContrpuntoCNC'  State= TRUE ;%{PE}%R 4.1.16,%MKUKATPBASIS,%COUT,%VOUTX,%P 2:11, 3:'OutRetroContrpuntoCNC', 5:TRUE, 6:
$OUT[11]=TRUE
;ENDFOLD
;FOLD WAIT FOR IN 13 'InContrpuntoAtrasCNC'  State= TRUE ;%{PE}%R 4.1.16,%MKUKATPBASIS,%CWAIT_FOR,%VWAIT_FOR,%P 1:0, 2:13, 3:'InContrpuntoAtrasCNC', 5:TRUE, 6:
WAIT FOR $IN[13]==TRUE
;ENDFOLD
;FOLD OUT 11 'OutRetroContrpuntoCNC'  State= FALSE ;%{PE}%R 4.1.16,%MKUKATPBASIS,%COUT,%VOUTX,%P 2:11, 3:'OutRetroContrpuntoCNC', 5:FALSE, 6:
$OUT[11]=FALSE
;ENDFOLD
;----------------

;--Cerrar Plato--
;FOLD OUT 8 'OutAbrirPlatoCNC'  State= FALSE ;%{PE}%R 4.1.16,%MKUKATPBASIS,%COUT,%VOUTX,%P 2:8, 3:'OutAbrirPlatoCNC', 5:FALSE, 6:
$OUT[8]=FALSE
;ENDFOLD
;FOLD OUT 9 'OutCerrarPlatoCNC'  State= TRUE ;%{PE}%R 4.1.16,%MKUKATPBASIS,%COUT,%VOUTX,%P 2:9, 3:'OutCerrarPlatoCNC', 5:TRUE, 6:
$OUT[9]=TRUE
;ENDFOLD
;FOLD WAIT FOR IN 15 'InPlatoCerradoCNC'  State= TRUE ;%{PE}%R 4.1.16,%MKUKATPBASIS,%CWAIT_FOR,%VWAIT_FOR,%P 1:0, 2:15, 3:'InPlatoCerradoCNC', 5:TRUE, 6:
WAIT FOR $IN[15]==TRUE
;ENDFOLD
;FOLD OUT 9 'OutCerrarPlatoCNC'  State= FALSE ;%{PE}%R 4.1.16,%MKUKATPBASIS,%COUT,%VOUTX,%P 2:9, 3:'OutCerrarPlatoCNC', 5:FALSE, 6:
$OUT[9]=FALSE
;ENDFOLD
;-----------------------

;--Cerrar Luneta--
;FOLD OUT 12 'OutAbrirLunetaCNC'  State= TRUE ;%{PE}%R 4.1.16,%MKUKATPBASIS,%COUT,%VOUTX,%P 2:12, 3:'OutAbrirLunetaCNC', 5:TRUE, 6:
$OUT[12]=TRUE
;ENDFOLD
;FOLD OUT 17 'OutCerrarLunetaCNC'  State= FALSE ;%{PE}%R 4.1.16,%MKUKATPBASIS,%COUT,%VOUTX,%P 2:17, 3:'OutCerrarLunetaCNC', 5:FALSE, 6:
$OUT[17]=FALSE
;ENDFOLD
;FOLD WAIT FOR IN 16 'InLunetaAbiertaCNC'  State= TRUE ;%{PE}%R 4.1.16,%MKUKATPBASIS,%CWAIT_FOR,%VWAIT_FOR,%P 1:0, 2:16, 3:'InLunetaAbiertaCNC', 5:TRUE, 6:
WAIT FOR $IN[16]==TRUE
;ENDFOLD
;FOLD OUT 12 'OutAbrirLunetaCNC'  State= FALSE ;%{PE}%R 4.1.16,%MKUKATPBASIS,%COUT,%VOUTX,%P 2:12, 3:'OutAbrirLunetaCNC', 5:FALSE, 6:
$OUT[12]=FALSE
;ENDFOLD
;FOLD WAIT Time= 1 sec;%{PE}%R 4.1.16,%MKUKATPBASIS,%CWAIT,%VWAIT,%P 2:1
WAIT SEC 1
;ENDFOLD
;-----------------

;FOLD SET Pinza1  State= OPN  Abrir;%{PE}%R 4.1.4,%MKUKATPGRP,%CGRP,%VGRP,%P 2:1, 4:1, 5:#NO, 6:Abrir, 8:0, 10:1
H50(GRP,1,1,GAbrir)
;ENDFOLD

;FOLD LIN Sal1_CNC CONT Vel= 2 m/s CPDAT12 Tool[1]:Tool1      Base[0];%{PE}%R 4.1.7,%MKUKATPBASIS,%CMOVE,%VLIN,%P 1:LIN, 2:Sal1_CNC, 3:C_DIS, 5:2, 7:CPDAT12
$BWDSTART = FALSE
LDAT_ACT=LCPDAT12
BAS(#CP_DAT)
FDAT_ACT=FSal1_CNC
BAS(#FRAMES)
BAS(#VEL_CP,2)
LIN XSal1_CNC C_DIS
;ENDFOLD
;FOLD PTP Sal2_CNC CONT Vel= 100 % PDAT24 Tool[1]:Tool1      Base[0];%{PE}%R 4.1.7,%MKUKATPBASIS,%CMOVE,%VPTP,%P 1:PTP, 2:Sal2_CNC, 3:C_PTP, 5:100, 7:PDAT24
$BWDSTART = FALSE
PDAT_ACT=PPDAT24
BAS(#PTP_DAT)
FDAT_ACT=FSal2_CNC
BAS(#FRAMES)
BAS(#VEL_PTP,100)
PTP XSal2_CNC C_PTP
;ENDFOLD
;FOLD PTP Sal3_CNC CONT Vel= 100 % PDAT1 Tool[1]:Tool1      Base[0];%{PE}%R 4.1.7,%MKUKATPBASIS,%CMOVE,%VPTP,%P 1:PTP, 2:Sal3_CNC, 3:C_PTP, 5:100, 7:PDAT1
$BWDSTART = FALSE
PDAT_ACT=PPDAT1
BAS(#PTP_DAT)
FDAT_ACT=FSal3_CNC
BAS(#FRAMES)
BAS(#VEL_PTP,100)
PTP XSal3_CNC C_PTP
;ENDFOLD

;----------------------------------------------------------

;FOLD PTP a CONT Vel= 100 % PDAT1 Tool[0] Base[0];%{PE}%R 4.1.7,%MKUKATPBASIS,%CMOVE,%VPTP,%P 1:PTP, 2:a, 3:C_PTP, 5:100, 7:PDAT1
$BWDSTART = FALSE
PDAT_ACT=PPDAT1
BAS(#PTP_DAT)
FDAT_ACT=Fa
BAS(#FRAMES)
BAS(#VEL_PTP,100)
PTP Xa C_PTP
;ENDFOLD

;FOLD PTP b CONT Vel= 50 % PDAT25 Tool[0] Base[0];%{PE}%R 4.1.7,%MKUKATPBASIS,%CMOVE,%VPTP,%P 1:PTP, 2:b, 3:C_PTP, 5:50, 7:PDAT25
$BWDSTART = FALSE
PDAT_ACT=PPDAT25
BAS(#PTP_DAT)
FDAT_ACT=Fb
BAS(#FRAMES)
BAS(#VEL_PTP,50)
PTP Xb C_PTP
;ENDFOLD
;FOLD WAIT Time=0 sec;%{PE}%R 5.5.33,%MKUKATPBASIS,%CWAIT,%VWAIT,%P 2:0
WAIT SEC 0
;ENDFOLD
;FOLD OUT 3 'OutRobotDentroCNC'  State= FALSE ;%{PE}%R 4.1.7,%MKUKATPBASIS,%COUT,%VOUTX,%P 2:3, 3:'OutRobotDentroCNC', 5:FALSE, 6:
$OUT[3]=FALSE
;ENDFOLD
;FOLD OUT 7 'OutRobotFuerCNC'  State= TRUE ;%{PE}%R 4.1.7,%MKUKATPBASIS,%COUT,%VOUTX,%P 2:7, 3:'OutRobotFuerCNC', 5:TRUE, 6:
$OUT[7]=TRUE
;ENDFOLD
;FOLD WAIT Time= 0 sec;%{PE}%R 4.1.7,%MKUKATPBASIS,%CWAIT,%VWAIT,%P 2:0
WAIT SEC 0
;ENDFOLD
;FOLD WAIT FOR IN 25 'InConRobotCNC'  State= TRUE CONT;%{PE}%R 4.1.7,%MKUKATPBASIS,%CWAIT_FOR,%VWAIT_FOR,%P 1:0, 2:25, 3:'InConRobotCNC', 5:TRUE, 6:CONTINUE
CONTINUE
WAIT FOR $IN[25]==TRUE
;ENDFOLD
;FOLD PULSE 2 'OutMarchaCNC'  State= TRUE   Time= 0.5 sec;%{PE}%R 4.1.7,%MKUKATPBASIS,%COUT,%VPULSE,%P 2:2, 3:'OutMarchaCNC', 5:TRUE, 6:, 8:0.5
PULSE($OUT[2], TRUE,0.5)
;ENDFOLD
;FOLD WAIT FOR IN 26 'InPuertaAbiertaCNC'  State= FALSE ;%{PE}%R 4.1.7,%MKUKATPBASIS,%CWAIT_FOR,%VWAIT_FOR,%P 1:0, 2:26, 3:'InPuertaAbiertaCNC', 5:FALSE, 6:
WAIT FOR $IN[26]==FALSE
;ENDFOLD

;FOLD PTP Frente_de_cinta CONT Vel= 40 % PDAT20 Tool[0] Base[0];%{PE}%R 4.1.7,%MKUKATPBASIS,%CMOVE,%VPTP,%P 1:PTP, 2:Frente_de_cinta, 3:C_PTP, 5:40, 7:PDAT20
$BWDSTART = FALSE
PDAT_ACT=PPDAT20
BAS(#PTP_DAT)
FDAT_ACT=FFrente_de_cinta
BAS(#FRAMES)
BAS(#VEL_PTP,40)
PTP XFrente_de_cinta C_PTP
;ENDFOLD

;ENDFOLD

;FOLD DEJAR PIEZA EN CINTA

;$OV_PRO=nVeloFuera
;FOLD PTP FrenteCintaNuevo CONT Vel= 30 % PDAT26 Tool[0] Base[0];%{PE}%R 4.1.16,%MKUKATPBASIS,%CMOVE,%VPTP,%P 1:PTP, 2:FrenteCintaNuevo, 3:C_PTP, 5:30, 7:PDAT26
$BWDSTART = FALSE
PDAT_ACT=PPDAT26
BAS(#PTP_DAT)
FDAT_ACT=FFrenteCintaNuevo
BAS(#FRAMES)
BAS(#VEL_PTP,30)
PTP XFrenteCintaNuevo C_PTP
;ENDFOLD

;FOLD PTP Aprox1_DejarCintaNuevo CONT Vel= 30 % PDAT27 Tool[2]:Tool2      Base[0];%{PE}%R 4.1.16,%MKUKATPBASIS,%CMOVE,%VPTP,%P 1:PTP, 2:Aprox1_DejarCintaNuevo, 3:C_PTP, 5:30, 7:PDAT27
$BWDSTART = FALSE
PDAT_ACT=PPDAT27
BAS(#PTP_DAT)
FDAT_ACT=FAprox1_DejarCintaNuevo
BAS(#FRAMES)
BAS(#VEL_PTP,30)
PTP XAprox1_DejarCintaNuevo C_PTP
;ENDFOLD

;FOLD LIN DejarCintaNuevo CONT Vel= 0.3 m/s CPDAT1 Tool[2]:Tool2      Base[0];%{PE}%R 4.1.16,%MKUKATPBASIS,%CMOVE,%VLIN,%P 1:LIN, 2:DejarCintaNuevo, 3:C_DIS, 5:0.3, 7:CPDAT1
$BWDSTART = FALSE
LDAT_ACT=LCPDAT1
BAS(#CP_DAT)
FDAT_ACT=FDejarCintaNuevo
BAS(#FRAMES)
BAS(#VEL_CP,0.3)
LIN XDejarCintaNuevo C_DIS
;ENDFOLD

;FOLD SET Pinza2  State= OPN  Abrir;%{PE}%R 4.1.4,%MKUKATPGRP,%CGRP,%VGRP,%P 2:2, 4:1, 5:#NO, 6:Abrir, 8:0, 10:1
H50(GRP,2,1,GAbrir)
;ENDFOLD

;FOLD PTP Aprox1_DejarCintaNuevo CONT Vel= 30 % PDAT27 Tool[2]:Tool2      Base[0];%{PE}%R 4.1.16,%MKUKATPBASIS,%CMOVE,%VPTP,%P 1:PTP, 2:Aprox1_DejarCintaNuevo, 3:C_PTP, 5:30, 7:PDAT27
$BWDSTART = FALSE
PDAT_ACT=PPDAT27
BAS(#PTP_DAT)
FDAT_ACT=FAprox1_DejarCintaNuevo
BAS(#FRAMES)
BAS(#VEL_PTP,30)
PTP XAprox1_DejarCintaNuevo C_PTP
;ENDFOLD

;FOLD PTP FrenteCintaNuevo CONT Vel= 30 % PDAT26 Tool[0] Base[0];%{PE}%R 4.1.16,%MKUKATPBASIS,%CMOVE,%VPTP,%P 1:PTP, 2:FrenteCintaNuevo, 3:C_PTP, 5:30, 7:PDAT26
$BWDSTART = FALSE
PDAT_ACT=PPDAT26
BAS(#PTP_DAT)
FDAT_ACT=FFrenteCintaNuevo
BAS(#FRAMES)
BAS(#VEL_PTP,30)
PTP XFrenteCintaNuevo C_PTP
;ENDFOLD



;ENDFOLD
;FOLD GESTION DE CICLO

nContadorPiezas=nContadorPiezas+1

IF bParadaManiobra==TRUE THEN
;FOLD PTP HOME  Vel= 25 % DEFAULT;%{PE}%R 4.1.7,%MKUKATPBASIS,%CMOVE,%VPTP,%P 1:PTP, 2:HOME, 3:, 5:25, 7:DEFAULT
$BWDSTART = FALSE
PDAT_ACT=PDEFAULT
BAS(#PTP_DAT)
FDAT_ACT=FHOME
BAS(#FRAMES)
BAS(#VEL_PTP,25)
$H_POS=XHOME
PTP XHOME
;ENDFOLD
outPilotoMarcha=FALSE
HALT
bParadaManiobra=FALSE

ELSE

ENDIF

ENDLOOP


;ENDFOLD


END

--- prueba_gewindebolzen_.dat ---
&ACCESS RVP
&REL 19
&COMMENT M36x315+allen
&PARAM TEMPLATE = C:\KRC\Roboter\Template\vorgabe
&PARAM EDITMASK = *
DEFDAT  PRUEBA_GEWINDEBOLZEN_
;FOLD EXTERNAL DECLARATIONS;%{PE}%V3.2.0,%MKUKATPBASIS,%CEXT,%VCOMMON,%P
;FOLD BAS EXT;%{PE}%V3.2.0,%MKUKATPBASIS,%CEXT,%VEXT,%P
EXT  BAS (BAS_COMMAND  :IN,REAL  :IN )
DECL INT SUCCESS
;ENDFOLD
;FOLD A10 EXT;%{E}%V3.2.0,%MKUKATPARC,%CEXT,%VEXT,%P
EXT  A10 (A_CMD_T  :IN,A_STRT_T  :IN,A_WELD_T  :IN,A_END_T  :IN,INT  :IN )
;ENDFOLD
;FOLD A20 EXT;%{E}%V3.2.0,%MKUKATPA20,%CEXT,%VEXT,%P
EXT  A20 (INT  :IN,WELD_ST  :IN,WELD_FI  :IN,INT  :IN )
;ENDFOLD
;FOLD GRIPPER EXT;%{E}%V3.2.0,%MKUKATPGRIPPER,%CEXT,%VEXT,%P
EXT  H50 (INT  :IN,INT  :IN,INT  :IN,GRP_TYP  :IN )
;ENDFOLD
;FOLD SPOT EXT;%{E}%V3.2.0,%MKUKATPSPOT,%CEXT,%VEXT,%P
EXT  USERSPOT (S_COMMAND  :IN,SPOT_TYPE  :IN )
;ENDFOLD
;FOLD TOUCHSENSE EXT;%{E}%V3.2.0,%MKUKATPTS,%CEXT,%VEXT,%P
EXT  H70 (INT  :IN,SRCH_TYP_2  :OUT,E6POS  :IN,SRCH_TYP_3  :IN,SRCH_TYP_2  :IN,SRCH_TYP_2  :IN,SRCH_TYP_2  :IN,SRCH_TYP_2  :IN,SRCH_TYP_2  :IN,INT  :IN )
;ENDFOLD
;FOLD USER EXT;%{E}%V3.2.0,%MKUKATPUSER,%CEXT,%VEXT,%P
;Make here your modifications
;ENDFOLD
;ENDFOLD

DECL BASIS_SUGG_T LAST_BASIS={POINT1[] "AcercarDescargaNuevo    ",POINT2[] "AcercarDescargaNuevo    ",CP_PARAMS[] "CPDAT13                 ",PTP_PARAMS[] "PDAT28                  ",CONT[] "C_PTP                   ",CP_VEL[] "0.3                     ",PTP_VEL[] "30                      "}
DECL E6POS XFRENTECINTA={x 586.713501,y 475.164886,z 2277.23389,a 88.4521027,b -44.9880409,c -179.531097,s 2,t 43,e1 0.0,e2 0.0,e3 0.0,e4 0.0,e5 0.0,e6 0.0}
DECL FDAT FFrenteCinta={TOOL_NO 0,BASE_NO 0,IPO_FRAME #BASE}
DECL PDAT PPDAT1={VEL 100.0,ACC 100.0,APO_DIST 90.0}
DECL FDAT FFrenteCNC={TOOL_NO 0,BASE_NO 0,IPO_FRAME #BASE}
DECL E6POS XDEJARPINZA2CINTA={x 1620.00403,y -0.00337643898,z 1909.99402,a -110.582497,b 89.9985199,c -110.582397,s 2,t 2,e1 0.0,e2 0.0,e3 0.0,e4 0.0,e5 0.0,e6 0.0}
DECL FDAT FDejarPinza2Cinta={TOOL_NO 2,BASE_NO 0,IPO_FRAME #BASE}
DECL PDAT PPDAT2={VEL 100.0,ACC 100.0,APO_DIST 100.0}
DECL E6POS XDEJARPINZA1CINTA={x -1031.74695,y 1452.62402,z 1168.32495,a 4.45051813,b 43.6923103,c -176.309998,s 2,t 35,e1 0.0,e2 0.0,e3 0.0,e4 0.0,e5 0.0,e6 0.0}
DECL FDAT FDejarPinza1Cinta={TOOL_NO 1,BASE_NO 0,IPO_FRAME #BASE}
DECL PDAT PPDAT3={VEL 100.0,ACC 100.0,APO_DIST 100.0}
DECL E6POS XENT1_COGERCINTA={x 444.522186,y 912.39978,z 1228.745,a 87.1254272,b -7.41709614,c -179.732895,s 2,t 43,e1 0.0,e2 0.0,e3 0.0,e4 0.0,e5 0.0,e6 0.0}
DECL FDAT FEnt1_CogerCinta={TOOL_NO 1,BASE_NO 0,IPO_FRAME #BASE}
DECL PDAT PPDAT4={VEL 100.0,ACC 100.0,APO_DIST 100.0}
DECL E6POS XENT2_COGERCINTA={x 241.129395,y 1260.59204,z 988.740173,a 89.6321411,b -16.7830791,c -179.436096,s 2,t 43,e1 0.0,e2 0.0,e3 0.0,e4 0.0,e5 0.0,e6 0.0}
DECL FDAT FEnt2_CogerCinta={TOOL_NO 1,BASE_NO 0,IPO_FRAME #BASE}
DECL PDAT PPDAT5={VEL 100.0,ACC 100.0,APO_DIST 100.0}
DECL E6POS XENT3COGERCINTA={x 240.920807,y 1266.87,z 965.138611,a 89.6319122,b -16.7829304,c -179.435501,s 2,t 43,e1 0.0,e2 0.0,e3 0.0,e4 0.0,e5 0.0,e6 0.0}
DECL FDAT FEnt3CogerCinta={TOOL_NO 1,BASE_NO 0,IPO_FRAME #BASE}
DECL PDAT PPDAT6={VEL 100.0,ACC 100.0,APO_DIST 100.0}
DECL LDAT LCPDAT1={VEL 2.0,ACC 100.0,APO_DIST 100.0,APO_FAC 50.0}
DECL E6POS XCOGERCINTA={x 240.621902,y 1277.82495,z 928.83667,a 89.6319427,b -16.7831707,c -179.435699,s 2,t 43,e1 0.0,e2 0.0,e3 0.0,e4 0.0,e5 0.0,e6 0.0}
DECL FDAT FCogerCinta={TOOL_NO 1,BASE_NO 0,IPO_FRAME #BASE}
DECL LDAT LCPDAT2={VEL 2.0,ACC 100.0,APO_DIST 100.0,APO_FAC 50.0}
DECL E6POS XSAL1_COGERCINTA={x 243.320999,y 1180.21704,z 1252.396,a 89.6317062,b -16.7828197,c -179.435501,s 2,t 43,e1 0.0,e2 0.0,e3 0.0,e4 0.0,e5 0.0,e6 0.0}
DECL FDAT FSal1_CogerCinta={TOOL_NO 1,BASE_NO 0,IPO_FRAME #BASE}
DECL LDAT LCPDAT3={VEL 2.0,ACC 100.0,APO_DIST 100.0,APO_FAC 50.0}
DECL E6POS XSAL2_COGERCINTA={x 303.099487,y 1180.77197,z 1267.77295,a 90.0943909,b -16.8520508,c -179.833298,s 2,t 43,e1 0.0,e2 0.0,e3 0.0,e4 0.0,e5 0.0,e6 0.0}
DECL FDAT FSal2_CogerCinta={TOOL_NO 1,BASE_NO 0,IPO_FRAME #BASE}
DECL PDAT PPDAT7={VEL 100.0,ACC 100.0,APO_DIST 100.0}
DECL E6POS XENT1_COGERCNC={x 1641.49902,y -669.381226,z 1323.13501,a 0.882562876,b -62.4571991,c -179.163101,s 2,t 42,e1 0.0,e2 0.0,e3 0.0,e4 0.0,e5 0.0,e6 0.0}
DECL FDAT FEnt1_CogerCNC={TOOL_NO 2,BASE_NO 0,IPO_FRAME #BASE}
DECL PDAT PPDAT8={VEL 100.0,ACC 100.0,APO_DIST 100.0}
DECL E6POS XENT2_COGERCNC={x 1641.49902,y -669.381226,z 1323.13501,a 0.882562876,b -62.4571991,c -179.163101,s 2,t 42,e1 0.0,e2 0.0,e3 0.0,e4 0.0,e5 0.0,e6 0.0}
DECL FDAT FEnt2_CogerCNC={TOOL_NO 2,BASE_NO 0,IPO_FRAME #BASE}
DECL PDAT PPDAT9={VEL 100.0,ACC 100.0,APO_DIST 100.0}
DECL E6POS XENT3_COGERCNC={x 1641.49902,y -669.381226,z 1323.13501,a 0.882562876,b -62.4571991,c -179.163101,s 2,t 42,e1 0.0,e2 0.0,e3 0.0,e4 0.0,e5 0.0,e6 0.0}
DECL FDAT FEnt3_CogerCNC={TOOL_NO 2,BASE_NO 0,IPO_FRAME #BASE}
DECL LDAT LCPDAT4={VEL 2.0,ACC 100.0,APO_DIST 100.0,APO_FAC 50.0}
DECL E6POS XCOGERCNC={x 2119.34106,y -572.075378,z 1077.37305,a 0.888575017,b -62.4623489,c -179.168503,s 2,t 42,e1 0.0,e2 0.0,e3 0.0,e4 0.0,e5 0.0,e6 0.0}
DECL FDAT FCogerCNC={TOOL_NO 2,BASE_NO 0,IPO_FRAME #BASE}
DECL LDAT LCPDAT5={VEL 2.0,ACC 100.0,APO_DIST 100.0,APO_FAC 50.0}
DECL E6POS XSAL1_COGERCNC={x 2121.07495,y -726.080627,z 1073.29199,a 0.886725187,b -62.4649506,c -179.165894,s 2,t 42,e1 0.0,e2 0.0,e3 0.0,e4 0.0,e5 0.0,e6 0.0}
DECL FDAT FSal1_CogerCNC={TOOL_NO 2,BASE_NO 0,IPO_FRAME #BASE}
DECL LDAT LCPDAT6={VEL 2.0,ACC 100.0,APO_DIST 100.0,APO_FAC 50.0}
DECL E6POS XSAL2_COGERCNC={x 2184.98901,y -732.532471,z 1085.38403,a 0.883620083,b -62.4613495,c -179.162704,s 2,t 42,e1 0.0,e2 0.0,e3 0.0,e4 0.0,e5 0.0,e6 0.0}
DECL FDAT FSal2_CogerCNC={TOOL_NO 2,BASE_NO 0,IPO_FRAME #BASE}
DECL LDAT LCPDAT7={VEL 2.0,ACC 100.0,APO_DIST 100.0,APO_FAC 50.0}
DECL E6POS XENT1_DEJARCNC={x 1919.52405,y -741.191895,z 1246.82703,a 0.568478525,b -35.9420815,c 179.852402,s 2,t 42,e1 0.0,e2 0.0,e3 0.0,e4 0.0,e5 0.0,e6 0.0}
DECL FDAT FEnt1_DejarCNC={TOOL_NO 1,BASE_NO 0,IPO_FRAME #BASE}
DECL PDAT PPDAT10={VEL 100.0,ACC 100.0,APO_DIST 100.0}
DECL E6POS XENT2_DEJARCNC={x 1919.52405,y -741.191895,z 1246.82703,a 0.568478525,b -35.9420815,c 179.852402,s 2,t 42,e1 0.0,e2 0.0,e3 0.0,e4 0.0,e5 0.0,e6 0.0}
DECL FDAT FEnt2_DejarCNC={TOOL_NO 1,BASE_NO 0,IPO_FRAME #BASE}
DECL PDAT PPDAT11={VEL 100.0,ACC 100.0,APO_DIST 100.0}
DECL E6POS XENT3_DEJARCNC={x 2118.04199,y -659.851929,z 1057.76196,a 1.58157098,b -55.0662117,c -179.354507,s 2,t 42,e1 0.0,e2 0.0,e3 0.0,e4 0.0,e5 0.0,e6 0.0}
DECL FDAT FEnt3_DejarCNC={TOOL_NO 1,BASE_NO 0,IPO_FRAME #BASE}
DECL LDAT LCPDAT8={VEL 2.0,ACC 100.0,APO_DIST 100.0,APO_FAC 50.0}
DECL E6POS XDEJARCNC={x 2118.03003,y -609.8573,z 1057.76294,a 1.58195102,b -55.0663681,c -179.354202,s 2,t 42,e1 0.0,e2 0.0,e3 0.0,e4 0.0,e5 0.0,e6 0.0}
DECL FDAT FDejarCNC={TOOL_NO 1,BASE_NO 0,IPO_FRAME #BASE}
DECL LDAT LCPDAT9={VEL 2.0,ACC 100.0,APO_DIST 100.0,APO_FAC 50.0}
DECL E6POS XSAL1_CNC={x 1597.93298,y -758.07782,z 1310.026,a 2.32089591,b -37.4369202,c 179.928894,s 2,t 42,e1 0.0,e2 0.0,e3 0.0,e4 0.0,e5 0.0,e6 0.0}
DECL FDAT FSal1_CNC={TOOL_NO 1,BASE_NO 0,IPO_FRAME #BASE}
DECL LDAT LCPDAT10={VEL 2.0,ACC 100.0,APO_DIST 100.0,APO_FAC 50.0}
DECL E6POS XSAL2_CNC={x 1597.93298,y -758.07782,z 1310.026,a 2.32089591,b -37.4369202,c 179.928894,s 2,t 42,e1 0.0,e2 0.0,e3 0.0,e4 0.0,e5 0.0,e6 0.0}
DECL FDAT FSal2_CNC={TOOL_NO 1,BASE_NO 0,IPO_FRAME #BASE}
DECL PDAT PPDAT12={VEL 100.0,ACC 100.0,APO_DIST 100.0}
DECL E6POS XSAL3_CNC={x 1597.93298,y -758.07782,z 1310.026,a 2.32089591,b -37.4369202,c 179.928894,s 2,t 42,e1 0.0,e2 0.0,e3 0.0,e4 0.0,e5 0.0,e6 0.0}
DECL FDAT FSal3_CNC={TOOL_NO 1,BASE_NO 0,IPO_FRAME #BASE}
DECL PDAT PPDAT13={VEL 100.0,ACC 100.0,APO_DIST 100.0}
DECL PDAT PPDAT14={VEL 100.0,ACC 100.0,APO_DIST 100.0}
DECL E6POS XENT1_DEJARCINTA={x -732.870728,y 1158.88794,z 2270.01904,a 59.0703812,b -89.6684494,c -91.9009628,s 2,t 43,e1 0.0,e2 0.0,e3 0.0,e4 0.0,e5 0.0,e6 0.0}
DECL FDAT FEnt1_DejarCinta={TOOL_NO 2,BASE_NO 0,IPO_FRAME #BASE}
DECL PDAT PPDAT15={VEL 100.0,ACC 100.0,APO_DIST 100.0}
DECL E6POS XENT2_DEJARCINTA={x -1001.48102,y 1524.125,z 1379.88904,a -179.701401,b -42.7616196,c 178.789902,s 2,t 35,e1 0.0,e2 0.0,e3 0.0,e4 0.0,e5 0.0,e6 0.0}
DECL FDAT FEnt2_DejarCinta={TOOL_NO 2,BASE_NO 0,IPO_FRAME #BASE}
DECL PDAT PPDAT16={VEL 100.0,ACC 100.0,APO_DIST 100.0}
DECL E6POS XSAL1_DEJARCINTA={x -732.870728,y 1158.88794,z 2270.01904,a 59.0703812,b -89.6684494,c -91.9009628,s 2,t 43,e1 0.0,e2 0.0,e3 0.0,e4 0.0,e5 0.0,e6 0.0}
DECL FDAT FSal1_DejarCinta={TOOL_NO 2,BASE_NO 0,IPO_FRAME #BASE}
DECL PDAT PPDAT17={VEL 100.0,ACC 100.0,APO_DIST 100.0}
DECL GRP_SUGG_T LAST_GRP={NUMBER[] "2                       ",STATE[] "1                       ",PARAMS[] "GDAT7                   "}
DECL GRP_TYP GGDAT0={G_APO #NO,TIME 0.200000003,CTRL #OFF,DLY 0,DST 1}
DECL GRP_TYP GGDAT2={G_APO #NO,TIME 0.200000003,CTRL #OFF,DLY 0,DST 1}
DECL GRP_TYP GGDAT3={G_APO #NO,TIME 0.200000003,CTRL #OFF,DLY 0,DST 1}
DECL GRP_TYP GCONT={G_APO #YES,TIME 0.0,CTRL #OFF,DLY 0,DST 0}
DECL GRP_TYP GGDAT4={G_APO #NO,TIME 0.200000003,CTRL #OFF,DLY 0,DST 1}
DECL GRP_TYP GGDAT5={G_APO #NO,TIME 0.200000003,CTRL #OFF,DLY 0,DST 1}
DECL GRP_TYP GGDAT6={G_APO #NO,TIME 0.200000003,CTRL #OFF,DLY 0,DST 1}
DECL GRP_TYP GGDAT7={G_APO #NO,TIME 0.200000003,CTRL #OFF,DLY 0,DST 1}
DECL GRP_TYP GCerrar={G_APO #NO,TIME 2.0,CTRL #OFF,DLY 0,DST 1}
DECL GRP_TYP GAbrir={G_APO #NO,TIME 1.0,CTRL #ON,DLY 0,DST 1}
DECL E6POS XSAL3_COJERCNC={x 2086.37598,y -737.606018,z 2293.60596,a -179.682907,b -54.0576591,c 0.203526199,s 2,t 42,e1 0.0,e2 0.0,e3 0.0,e4 0.0,e5 0.0,e6 0.0}
DECL FDAT FSal3_CojerCNC={TOOL_NO 2,BASE_NO 0,IPO_FRAME #BASE}
DECL LDAT LCPDAT11={VEL 2.0,ACC 100.0,APO_DIST 100.0,APO_FAC 50.0}
DECL E6POS XENT1DEJARCINTA={x -732.877625,y 1158.89099,z 2270.01294,a 59.1002197,b -89.6681366,c -91.9304428,s 2,t 43,e1 0.0,e2 0.0,e3 0.0,e4 0.0,e5 0.0,e6 0.0}
DECL FDAT FEnt1DejarCinta={TOOL_NO 2,BASE_NO 0,IPO_FRAME #BASE}
DECL E6POS XDEJARCINTA={x 170.750595,y -2731.46899,z 1167.23706,a -85.0863037,b -59.3405418,c 177.517303,s 2,t 34,e1 0.0,e2 0.0,e3 0.0,e4 0.0,e5 0.0,e6 0.0}
DECL FDAT FDejarCinta={TOOL_NO 2,BASE_NO 0,IPO_FRAME #BASE}
DECL E6POS XDejar1Pinza1Cinta={x -186.125397,y 753.741089,z 1449.41602,a 95.8809891,b 44.9203796,c -173.800201,s 2,t 43,e1 0.0,e2 0.0,e3 0.0,e4 0.0,e5 0.0,e6 0.0}
DECL FDAT FDejar1Pinza1Cinta={TOOL_NO 1,BASE_NO 0,IPO_FRAME #BASE}
DECL E6POS XDEJAR11PINZA1CINTA={x 8.99515533,y 1556.49805,z 1254.88403,a -178.753204,b 22.3286991,c -179.640305,s 2,t 43,e1 0.0,e2 0.0,e3 0.0,e4 0.0,e5 0.0,e6 0.0}
DECL FDAT FDejar11Pinza1Cinta={TOOL_NO 1,BASE_NO 0,IPO_FRAME #BASE}
DECL PDAT PPDAT18={VEL 100.0,ACC 100.0,APO_DIST 100.0}
DECL E6POS XDejar12Pinza1Cinta={x -186.133896,y 753.739807,z 1449.41504,a 95.8812408,b 44.9207687,c -173.7995,s 2,t 43,e1 0.0,e2 0.0,e3 0.0,e4 0.0,e5 0.0,e6 0.0}
DECL FDAT FDejar12Pinza1Cinta={TOOL_NO 1,BASE_NO 0,IPO_FRAME #BASE}
DECL E6POS XDEJAR13PINZA1CINTA={x -1031.74597,y 1452.62195,z 1331.95105,a 4.45047188,b 43.6921806,c -176.310303,s 2,t 35,e1 0.0,e2 0.0,e3 0.0,e4 0.0,e5 0.0,e6 0.0}
DECL FDAT FDejar13Pinza1Cinta={TOOL_NO 1,BASE_NO 0,IPO_FRAME #BASE}
DECL E6POS XDEJAR14PINZA1CINTA={x -822.157227,y 1482.88794,z 1540.41504,a 46.40839,b 58.6334381,c -133.363007,s 2,t 43,e1 0.0,e2 0.0,e3 0.0,e4 0.0,e5 0.0,e6 0.0}
DECL FDAT FDejar14Pinza1Cinta={TOOL_NO 1,BASE_NO 0,IPO_FRAME #BASE}
DECL PDAT PPDAT19={VEL 100.0,ACC 100.0,APO_DIST 100.0}
DECL FDAT FFrenteaCNC={TOOL_NO 0,BASE_NO 0,IPO_FRAME #BASE}
DECL E6POS XFRENTE_DE_CNC={x 974.234619,y -690.713074,z 1679.229,a 1.502931,b -17.4592896,c -179.594299,s 2,t 42,e1 0.0,e2 0.0,e3 0.0,e4 0.0,e5 0.0,e6 0.0}
DECL FDAT FFrente_de_cnc={TOOL_NO 0,BASE_NO 0,IPO_FRAME #BASE}
DECL E6POS XP0={x 1108.72595,y -726.085205,z 753.8255,a -0.460143209,b 27.5578899,c 178.797806,s 2,t 42,e1 0.0,e2 0.0,e3 0.0,e4 0.0,e5 0.0,e6 0.0}
DECL E6POS XFRENTE_DE_CINTA={x 904.580627,y -822.965393,z 2173.77295,a 3.13468695,b -69.9075623,c 179.628098,s 2,t 42,e1 0.0,e2 0.0,e3 0.0,e4 0.0,e5 0.0,e6 0.0}
DECL FDAT FFrente_de_cinta={TOOL_NO 0,BASE_NO 0,IPO_FRAME #BASE}
DECL PDAT PPDAT20={VEL 100.0,ACC 100.0,APO_DIST 90.0}
DECL PDAT PPDAT21={VEL 100.0,ACC 100.0,APO_DIST 100.0}
DECL E6POS XA={x 1132.73206,y -775.992371,z 1906.48901,a 2.70289493,b -82.4367294,c 179.570999,s 2,t 42,e1 0.0,e2 0.0,e3 0.0,e4 0.0,e5 0.0,e6 0.0}
DECL FDAT Fa={TOOL_NO 0,BASE_NO 0,IPO_FRAME #BASE}
DECL PDAT PPDAT22={VEL 100.0,ACC 100.0,APO_DIST 90.0}
DECL PDAT PPDAT23={VEL 100.0,ACC 100.0,APO_DIST 90.0}
DECL PDAT PPDAT24={VEL 100.0,ACC 100.0,APO_DIST 90.0}
DECL LDAT LCPDAT12={VEL 2.0,ACC 100.0,APO_DIST 100.0,APO_FAC 50.0}
DECL PDAT PPDAT25={VEL 100.0,ACC 100.0,APO_DIST 90.0}
DECL E6POS Xb={x 1132.73206,y -775.992371,z 1906.48901,a 2.70289493,b -82.4367294,c 179.570999,s 2,t 42,e1 0.0,e2 0.0,e3 0.0,e4 0.0,e5 0.0,e6 0.0}
DECL FDAT Fb={TOOL_NO 0,BASE_NO 0,IPO_FRAME #BASE}
DECL E6POS XFRENTECINTANUEVO={x 80.9268265,y -1146.89099,z 1902.69604,a -87.2553864,b -36.0338211,c 178.546494,s 2,t 34,e1 0.0,e2 0.0,e3 0.0,e4 0.0,e5 0.0,e6 0.0}
DECL FDAT FFrenteCintaNuevo={TOOL_NO 0,BASE_NO 0,IPO_FRAME #BASE}
DECL PDAT PPDAT26={VEL 100.0,ACC 100.0,APO_DIST 100.0}
DECL E6POS XAPROX1_DEJARCINTANUEVO={x 170.7565,y -2731.43091,z 1356.33203,a -85.0873718,b -59.3369789,c 177.518402,s 2,t 34,e1 0.0,e2 0.0,e3 0.0,e4 0.0,e5 0.0,e6 0.0}
DECL FDAT FAprox1_DejarCintaNuevo={TOOL_NO 2,BASE_NO 0,IPO_FRAME #BASE}
DECL PDAT PPDAT27={VEL 100.0,ACC 100.0,APO_DIST 100.0}
DECL E6POS XDejarCintaNuevo={x 170.750595,y -2731.46899,z 1167.23706,a -85.0863037,b -59.3405418,c 177.517303,s 2,t 34,e1 0.0,e2 0.0,e3 0.0,e4 0.0,e5 0.0,e6 0.0}
DECL FDAT FDejarCintaNuevo={TOOL_NO 2,BASE_NO 0,IPO_FRAME #BASE}
DECL E6POS XACERCARDESCARGANUEVO={x 560.754272,y -203.6698,z 2916.69897,a 159.668304,b -9.53805161,c -0.595628381,s 6,t 58,e1 0.0,e2 0.0,e3 0.0,e4 0.0,e5 0.0,e6 0.0}
DECL FDAT FAcercarDescargaNuevo={TOOL_NO 0,BASE_NO 0,IPO_FRAME #BASE}
DECL PDAT PPDAT28={VEL 100.0,ACC 100.0,APO_DIST 100.0}
DECL E6POS XAPROX2_DEJARCINTANUEVO={x 204.782394,y -2509.16504,z 1812.34705,a 89.5281219,b -88.9469833,c 3.94414401,s 2,t 34,e1 0.0,e2 0.0,e3 0.0,e4 0.0,e5 0.0,e6 0.0}
DECL FDAT FAprox2_DejarCintaNuevo={TOOL_NO 2,BASE_NO 0,IPO_FRAME #BASE}
DECL PDAT PPDAT29={VEL 100.0,ACC 100.0,APO_DIST 100.0}
DECL E6POS XAPROX3_DEJARCINTANUEVO={x 205.497406,y -2481.12793,z 2466.38892,a 96.1354065,b -32.7504501,c -0.687986612,s 6,t 50,e1 0.0,e2 0.0,e3 0.0,e4 0.0,e5 0.0,e6 0.0}
DECL FDAT FAprox3_DejarCintaNuevo={TOOL_NO 2,BASE_NO 0,IPO_FRAME #BASE}
DECL PDAT PPDAT30={VEL 100.0,ACC 100.0,APO_DIST 100.0}
DECL E6POS XAPROX4_DEJARCINTANUEVO={x 205.494797,y -2481.10889,z 2194.96191,a 96.134903,b -32.7487793,c -0.687672615,s 6,t 50,e1 0.0,e2 0.0,e3 0.0,e4 0.0,e5 0.0,e6 0.0}
DECL FDAT FAprox4_DejarCintaNuevo={TOOL_NO 2,BASE_NO 0,IPO_FRAME #BASE}
DECL LDAT LCPDAT13={VEL 2.0,ACC 100.0,APO_DIST 100.0,APO_FAC 50.0}
ENDDAT
